INTERFACE ITF_TopElement_HMI

END_INTERFACE

(* stored: Version 1.1.0.1, ProductVersion 3.1.4024.15
   Itf ITF_TopElement_HMI: Id {3b91dccd-4a6c-4fc9-b449-5eb45f3b7186} *)
